// TIA Portal V16 export
// export: Created 2024-09-05T17:39:14.4873427Z, ExportSetting WithDefaults, DisplayName Totally Integrated Automation Portal, DisplayVersion V16 Update 6, DisplayName TIA Portal Version Control Interface, DisplayVersion V16 Update 2, DisplayName TIA Portal Openness, DisplayVersion V16 Update 6, DisplayName STEP 7 Professional, DisplayVersion V16 Update 6, DisplayName STEP 7 Safety, DisplayVersion V16, DisplayName WinCC Advanced, DisplayVersion V16 Update 6
DATA_BLOCK "DB_EksData"   // DB5052
{ S7_Optimized_Access := 'TRUE' }
VERSION : 0.1
// stored: AutoNumber false, DBAccessibleFromOPCUA true, IsOnlyStoredInLoadMemory false, IsRetainMemResEnabled false, IsWriteProtectedInAS false, MemoryReserve 0
   VAR
      EmptyKey { S7_SetPoint := 'True'} : "UDT_EksKey";
      LoadedData { S7_SetPoint := 'True'} : "UDT_EksKey";
      ActualKey { S7_SetPoint := 'True'} : "UDT_EksKey";
      LastKey { S7_SetPoint := 'True'} : "UDT_EksKey";
      KeyListHMI { S7_SetPoint := 'True'} : Array[1..10] of "UDT_EksKey";
   END_VAR
BEGIN
   EmptyKey.Level := 0;
   EmptyKey.EmployeeID[1..4] := ' ';
   EmptyKey.KeyID[1..16] := ' ';
   EmptyKey.Comment[1..20] := ' ';
   LoadedData.Level := 0;
   LoadedData.EmployeeID[1..4] := ' ';
   LoadedData.KeyID[1] := '0';
   LoadedData.KeyID[2] := '3';
   LoadedData.KeyID[3] := '7';
   LoadedData.KeyID[4] := '2';
   LoadedData.KeyID[5] := '4';
   LoadedData.KeyID[6] := '5';
   LoadedData.KeyID[7] := '2';
   LoadedData.KeyID[8] := '9';
   LoadedData.KeyID[9] := 'A';
   LoadedData.KeyID[10] := '6';
   LoadedData.KeyID[11..12] := '0';
   LoadedData.KeyID[13] := '1';
   LoadedData.KeyID[14] := '0';
   LoadedData.KeyID[15] := '3';
   LoadedData.KeyID[16] := '2';
   LoadedData.Comment[1..20] := ' ';
   ActualKey.Level := 5;
   ActualKey.EmployeeID[1..4] := ' ';
   ActualKey.KeyID[1] := '0';
   ActualKey.KeyID[2] := '3';
   ActualKey.KeyID[3] := '7';
   ActualKey.KeyID[4] := '2';
   ActualKey.KeyID[5] := '4';
   ActualKey.KeyID[6] := '5';
   ActualKey.KeyID[7] := '2';
   ActualKey.KeyID[8] := '9';
   ActualKey.KeyID[9] := 'A';
   ActualKey.KeyID[10] := '6';
   ActualKey.KeyID[11..12] := '0';
   ActualKey.KeyID[13] := '1';
   ActualKey.KeyID[14] := '0';
   ActualKey.KeyID[15] := '3';
   ActualKey.KeyID[16] := '2';
   ActualKey.Comment[1..20] := ' ';
   LastKey.Level := 0;
   LastKey.EmployeeID[1..4] := ' ';
   LastKey.KeyID[1..16] := ' ';
   LastKey.Comment[1..20] := ' ';
   KeyListHMI[1..10].Level := 0;
   KeyListHMI[1].EmployeeID[1..4] := ' ';
   KeyListHMI[2].EmployeeID[1..4] := ' ';
   KeyListHMI[3].EmployeeID[1..4] := ' ';
   KeyListHMI[4].EmployeeID[1..4] := ' ';
   KeyListHMI[5].EmployeeID[1..4] := ' ';
   KeyListHMI[6].EmployeeID[1..4] := ' ';
   KeyListHMI[7].EmployeeID[1..4] := ' ';
   KeyListHMI[8].EmployeeID[1..4] := ' ';
   KeyListHMI[9].EmployeeID[1..4] := ' ';
   KeyListHMI[10].EmployeeID[1..4] := ' ';
   KeyListHMI[1].KeyID[1..16] := ' ';
   KeyListHMI[2].KeyID[1..16] := ' ';
   KeyListHMI[3].KeyID[1..16] := ' ';
   KeyListHMI[4].KeyID[1..16] := ' ';
   KeyListHMI[5].KeyID[1..16] := ' ';
   KeyListHMI[6].KeyID[1..16] := ' ';
   KeyListHMI[7].KeyID[1..16] := ' ';
   KeyListHMI[8].KeyID[1..16] := ' ';
   KeyListHMI[9].KeyID[1..16] := ' ';
   KeyListHMI[10].KeyID[1..16] := ' ';
   KeyListHMI[1].Comment[1..20] := ' ';
   KeyListHMI[2].Comment[1..20] := ' ';
   KeyListHMI[3].Comment[1..20] := ' ';
   KeyListHMI[4].Comment[1..20] := ' ';
   KeyListHMI[5].Comment[1..20] := ' ';
   KeyListHMI[6].Comment[1..20] := ' ';
   KeyListHMI[7].Comment[1..20] := ' ';
   KeyListHMI[8].Comment[1..20] := ' ';
   KeyListHMI[9].Comment[1..20] := ' ';
   KeyListHMI[10].Comment[1..20] := ' ';
END_DATA_BLOCK
